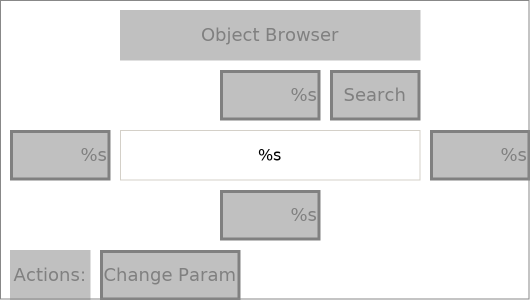
VISUALIZATION ObjectBrowser  // 530x300
VAR
	active_object: I_SYS_COMP_Object := _SYS_COMP_.object_list;
	
	search_name: STRING := 'Object';
	
	parent_name: STRING := '';
	child_name: STRING := '';
	
	next_object_name: STRING := '';
	prev_object_name: STRING := '';
	
END_VAR
    RoundedRectangle (120,10 300x50), "Object Browser"
    RoundedRectangle (10,130 100x50), "%s", text variable: CONCAT(prev_object_name, ' .')
        OnMouseUp: execute {
            IF active_object <> 0 AND_THEN active_object._SYS_COMP_prev_object <> 0 THEN
            	active_object := active_object._SYS_COMP_prev_object;
            	search_name := active_object.name;
            	IF active_object._SYS_COMP_parent <> 0 THEN
            		parent_name := active_object._SYS_COMP_parent.name;
            	ELSE
            		parent_name := 'Global Object.list';
            	END_IF
            	IF active_object._SYS_COMP_last_child <> 0 THEN
            		child_name := active_object._SYS_COMP_last_child.name;
            	ELSE
            		child_name := '';
            	END_IF
            	IF active_object._SYS_COMP_next_object <> 0 THEN
            		next_object_name := active_object._SYS_COMP_next_object.name;
            	ELSE
            		next_object_name := '';
            	END_IF
            	IF active_object._SYS_COMP_prev_object <> 0 THEN
            		prev_object_name := active_object._SYS_COMP_prev_object.name;
            	ELSE
            		prev_object_name := '';
            	END_IF
            END_IF
        }
    RoundedRectangle (430,130 100x50), "%s", text variable: CONCAT(next_object_name, ' .')
        OnMouseUp: execute {
            IF active_object <> 0 AND_THEN active_object._SYS_COMP_next_object <> 0 THEN
            	active_object := active_object._SYS_COMP_next_object;
            	search_name := active_object.name;
            	IF active_object._SYS_COMP_parent <> 0 THEN
            		parent_name := active_object._SYS_COMP_parent.name;
            	ELSE
            		parent_name := 'Global ObjectList';
            	END_IF
            	IF active_object._SYS_COMP_last_child <> 0 THEN
            		child_name := active_object._SYS_COMP_last_child.name;
            	ELSE
            		child_name := '';
            	END_IF
            	IF active_object._SYS_COMP_next_object <> 0 THEN
            		next_object_name := active_object._SYS_COMP_next_object.name;
            	ELSE
            		next_object_name := '';
            	END_IF
            	IF active_object._SYS_COMP_prev_object <> 0 THEN
            		prev_object_name := active_object._SYS_COMP_prev_object.name;
            	ELSE
            		prev_object_name := '';
            	END_IF
            END_IF
        }
    RoundedRectangle (220,190 100x50), "%s", text variable: CONCAT(child_name, ' .')
        OnMouseUp: execute {
            IF active_object <> 0 AND_THEN active_object._SYS_COMP_last_child <> 0 THEN
            	active_object := active_object._SYS_COMP_last_child;
            	search_name := active_object.name;
            	IF active_object._SYS_COMP_parent <> 0 THEN
            		parent_name := active_object._SYS_COMP_parent.name;
            	ELSE
            		parent_name := 'Global ObjectList';
            	END_IF
            	IF active_object._SYS_COMP_last_child <> 0 THEN
            		child_name := active_object._SYS_COMP_last_child.name;
            	ELSE
            		child_name := '';
            	END_IF
            	IF active_object._SYS_COMP_next_object <> 0 THEN
            		next_object_name := active_object._SYS_COMP_next_object.name;
            	ELSE
            		next_object_name := '';
            	END_IF
            	IF active_object._SYS_COMP_prev_object <> 0 THEN
            		prev_object_name := active_object._SYS_COMP_prev_object.name;
            	ELSE
            		prev_object_name := '';
            	END_IF
            END_IF
        }
    RoundedRectangle (220,70 100x50), "%s", text variable: CONCAT(parent_name, ' .')
        OnMouseUp: execute {
            IF active_object <> 0 AND_THEN active_object._SYS_COMP_parent <> 0 THEN
            	active_object := active_object._SYS_COMP_parent;
            	search_name := active_object.name;
            	IF active_object._SYS_COMP_parent <> 0 THEN
            		parent_name := active_object._SYS_COMP_parent.name;
            	ELSE
            		parent_name := 'Global ObjectList';
            	END_IF
            	IF active_object._SYS_COMP_last_child <> 0 THEN
            		child_name := active_object._SYS_COMP_last_child.name;
            	ELSE
            		child_name := '';
            	END_IF
            	IF active_object._SYS_COMP_next_object <> 0 THEN
            		next_object_name := active_object._SYS_COMP_next_object.name;
            	ELSE
            		next_object_name := '';
            	END_IF
            	IF active_object._SYS_COMP_prev_object <> 0 THEN
            		prev_object_name := active_object._SYS_COMP_prev_object.name;
            	ELSE
            		prev_object_name := '';
            	END_IF
            END_IF
        }
    Textfield (120,130 300x50), "%s", text variable: search_name
        OnMouseUp: write the text variable via Default
    RoundedRectangle (10,250 80x50), "Actions:"
    RoundedRectangle (100,250 140x50), "Change Param"
        OnMouseUp: OpenDialog Dialog=ParamDialog, Parameters={active_object: active_object, active_param: , name: , new_value: , value: }, OpenModal=True, OpenCentered=True
    RoundedRectangle (330,70 90x50), "Search"
        OnMouseUp: execute {
            active_object := _SYS_COMP_.Get_object(search_name);
            IF active_object <> 0 THEN
            	search_name := active_object.name;
            	IF active_object._SYS_COMP_parent <> 0 THEN
            		parent_name := active_object._SYS_COMP_parent.name;
            	ELSE
            		parent_name := 'Global ObjectList';
            	END_IF
            	IF active_object._SYS_COMP_last_child <> 0 THEN
            		child_name := active_object._SYS_COMP_last_child.name;
            	ELSE
            		child_name := '';
            	END_IF
            	IF active_object._SYS_COMP_next_object <> 0 THEN
            		next_object_name := active_object._SYS_COMP_next_object.name;
            	ELSE
            		next_object_name := '';
            	END_IF
            	IF active_object._SYS_COMP_prev_object <> 0 THEN
            		prev_object_name := active_object._SYS_COMP_prev_object.name;
            	ELSE
            		prev_object_name := '';
            	END_IF
            ELSE
            	search_name := 'OBJECT DOESNT EXIST';
            	parent_name := '';
            	child_name := '';
            	next_object_name := '';
            	prev_object_name := '';
            END_IF
        }
END_VISUALIZATION

(* stored: Version 1.1.0.1, ProductVersion 3.1.4024.12
   Visu ObjectBrowser: Id {d3117cb4-da8b-4fa8-a94d-fbe925c90c1c} *)
